TYPE Tc2_EtherCAT_Output_typ : 	
	STRUCT 
		Status 	: Tc2_EtherCAT_Statuses_typ;
		Error 	: Tc2_EtherCAT_Error_typ;
	END_STRUCT
END_TYPE

(* stored: Version 1.1.0.1, ProductVersion 3.1.4024.3
   DUT Tc2_EtherCAT_Output_typ: Id {a91734c3-cdf4-05dd-3963-305f08834b2c} *)
